VAR_GLOBAL CONSTANT
	iSLAVEADDR_ARR_SIZE: INT := 255;
END_VAR

(* stored: Version 1.1.0.1, ProductVersion 3.1.0.12
   GVL Globale_EtherCATDiag: Id {2998fef1-e645-4fd5-b5b6-42ac75b58c2f} *)
